(* CODESYS project Scheduler.project
   Company: Control Techniques
   Title: Scheduller
   Description: This program can be use to Start/stop motor  following  an weekly schedulle.  Up to 3 different time slices can be setup.
   Author: Angel Guerrero
   Version: 0.0.1

Project tree, tasks and I/O mapping:
  Drive : Unidrive M700, Nidec Control Techniques, version 1.8.0.9
    application Application
      Task Configuration
        Freewheeling
      program Freewheeling [ST]: TIMER, validate, get_vars, Initial
      function block Scheduler [ST]: Time_Check
      global variables GVL
      function Wait_Time [ST]
    RTEthernet
    Ethernet : Ethernet, Nidec Control Techniques, version 1.8.0.9
    <Empty>
    <Empty>
    <Empty>
  Advanced Link Editor
*)

// Drive/Application/GVL
{attribute 'qualified_only'}
VAR_GLOBAL
	RTC		 : DINT;  //RTC time from drive
	get_hr	 : UINT;  //Variable to hold hour 
	get_min	 : UINT;  //Variable to holf minutes [not used yet]
	get_sec	 : UINT;  //Variable that hold seconds [not used yet]
	get_wkd : SINT;  //Holds the week day
	enbl_mcr : INT;   //Enable Macro
END_VAR

// Drive/Application/Freewheeling
PROGRAM Freewheeling
VAR	
	err				: BOOL;			
	Scheduler_1		: Scheduler;
	Scheduler_2		: Scheduler;
	Scheduler_3		: Scheduler;	
	first_shoot		: BOOL := TRUE;	
END_VAR

//Version 0.00.01
//Angel Guerrero  Applications Engineer LatinAmerica July/2019
//============================================\\
get_vars();   	//Read RTC data
Initial();      //Macro setup
validate();   	//Validate setup data is correct
TIMER();        //Call the main program wich is timer.

ACTION TIMER:
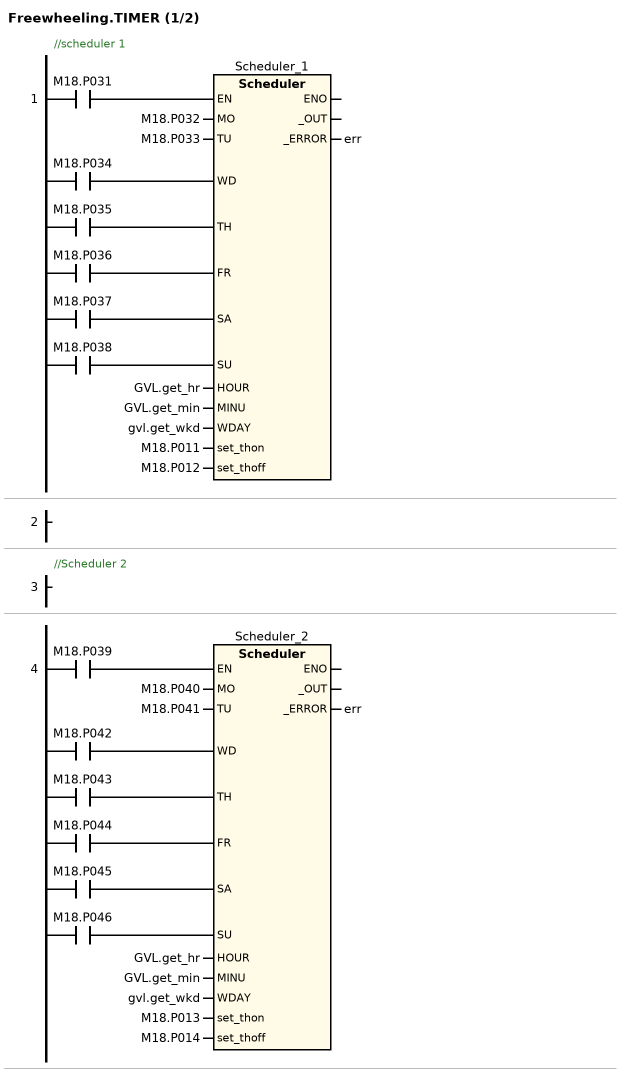
// NETWORK 1
// //scheduler 1
IF M18.P031 THEN
    Scheduler_1(
        MO := M18.P032,
        TU := M18.P033,
        WD := M18.P034,
        TH := M18.P035,
        FR := M18.P036,
        SA := M18.P037,
        SU := M18.P038,
        HOUR := GVL.get_hr,
        MINU := GVL.get_min,
        WDAY := gvl.get_wkd,
        set_thon := M18.P011,
        set_thoff := M18.P012,
        _ERROR => err); // Scheduler
END_IF

// NETWORK 2

// NETWORK 3
// //Scheduler 2

// NETWORK 4
IF M18.P039 THEN
    Scheduler_2(
        MO := M18.P040,
        TU := M18.P041,
        WD := M18.P042,
        TH := M18.P043,
        FR := M18.P044,
        SA := M18.P045,
        SU := M18.P046,
        HOUR := GVL.get_hr,
        MINU := GVL.get_min,
        WDAY := gvl.get_wkd,
        set_thon := M18.P013,
        set_thoff := M18.P014,
        _ERROR => err); // Scheduler
END_IF

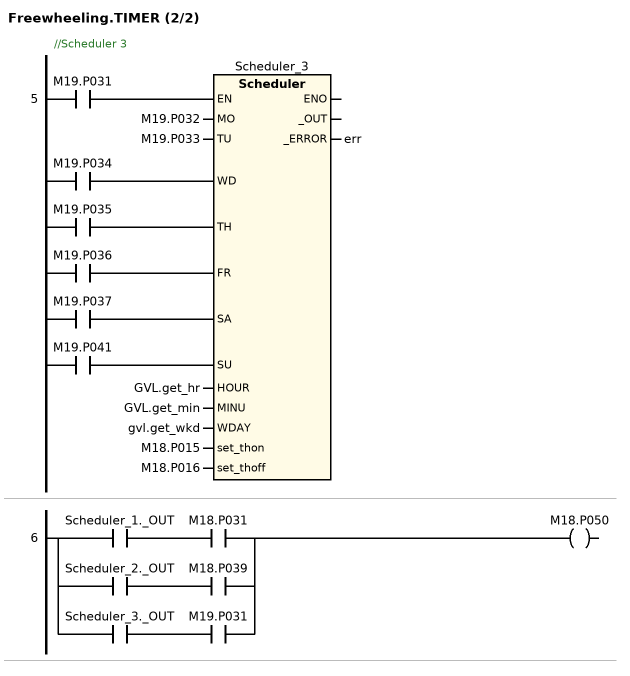
// NETWORK 5
// //Scheduler 3
IF M19.P031 THEN
    Scheduler_3(
        MO := M19.P032,
        TU := M19.P033,
        WD := M19.P034,
        TH := M19.P035,
        FR := M19.P036,
        SA := M19.P037,
        SU := M19.P041,
        HOUR := GVL.get_hr,
        MINU := GVL.get_min,
        WDAY := gvl.get_wkd,
        set_thon := M18.P015,
        set_thoff := M18.P016,
        _ERROR => err); // Scheduler
END_IF

// NETWORK 6
M18.P050 := Scheduler_1._OUT AND M18.P031 OR Scheduler_2._OUT AND M18.P039 OR Scheduler_3._OUT AND M19.P031;
END_ACTION

ACTION validate:
//Validate Scheduler 0 time ON/OFF is in correct range
IF M18.P011 >23 THEN
	M18.P011:=23;
END_IF
IF M18.P011 <0 THEN
	M18.P011:=0;
END_IF
//Validate Scheduler 0 time ON/OFF is in correct range
IF M18.P012 >23 THEN
	M18.P012:=23;
END_IF
IF M18.P012 <0 THEN
	M18.P012:=0;
END_IF
//Validate Scheduler 1 time ON/OFF is in correct range
IF M18.P013 >23 THEN
	M18.P013:=23;
END_IF
IF M18.P013 <0 THEN
	M18.P013:=0;
END_IF
//Validate Scheduler 1 time ON/OFF is in correct range
IF M18.P014 >23 THEN
	M18.P014:=23;
END_IF
IF M18.P014 <0 THEN
	M18.P014:=0;
END_IF
//Validate Scheduler 2 time ON/OFF is in correct range
IF M18.P015 >23 THEN
	M18.P015:=23;
END_IF
IF M18.P015 <0 THEN
	M18.P015:=0;
END_IF
//Validate Scheduler 2 time ON/OFF is in correct range
IF M18.P016 >23 THEN
	M18.P016:=23;
END_IF
IF M18.P016 <0 THEN
	M18.P016:=0;
END_IF
//Validate y Setup mode is 1 or 2 
IF M18.P030 >3 THEN
	M18.P030:=3;   //Remote Keypad
END_IF
IF M18.P030 <1 THEN
	M18.P030:=1;   //Local Keypad
END_IF
END_ACTION

ACTION get_vars:


gvl.RTC			:= M06.P017;                        			//Get time from RTC
gvl.get_hr  	:= DINT_TO_UINT(TRUNC(gvl.RTC/10000));  		//Get HRs
gvl.get_min 	:= DINT_TO_UINT((TRUNC(gvl.RTC/100)) MOD 100);  //Get Mins
gvl.get_sec 	:= DINT_TO_UINT((gvl.RTC) MOD 100);   			//seconds
gvl.enbl_mcr 	:= M18.P029;                                    // User Parameter to enter a "secret" value 1234  to deploy a Macro that prepare drive to link schduler output to Rfwd command
gvl.get_wkd     := M06.P018;                                    // get week day from Pr 06.P018
END_ACTION

ACTION Initial:
//macro to setup the  drive to start stop based on the scheduler
IF (gvl.enbl_mcr =1234 AND first_shoot=TRUE) THEN   	// If 1234 is set on Pr18.P029 then we accomodate drive parameters use the scheduller output for the rfwd command
	M08.P022	:=	0.00; 		//clear destination [default is M06.030] RunFwd
	M09.P004	:=	18.050;   	// Logic Fucntion 1 source1-->Asigns the Schduller ouput to the  funtion 
    M09.P006    :=  0.00;	    // Logic Function 1 Source 2-->we can probably get rid of this set to allow user add a DI to this source as way to stop the drive by any other condition
	M09.P007    :=  TRUE;       // Logic Function 1 Source 2 invert
	M09.P008    :=  FALSE;      // Logic Function 1 Output invert. 
	M09.P010    :=  6.030;      // Logic Funtion 1 Destination  set to Pr [6.030] RunFwd
	M10.P000	:=	1001;    	//Save Parameters
	M10.P038	:= 	100; 	 	//Reset Drive
	Wait_Time(T#400MS);         //Delay for 400ms after save and reset. 
	first_shoot := FALSE;       //Run this  section once once
	
END_IF

//Setup the source  to get the RTC from  Local Keypad or Remote .
//When mode is change user must save parameter manually and reset the drive
IF M18.P030=1 THEN 
	M06.P019:=4;     //M18.P030=4  Local Keypad
	ELSIF  M18.P030=2 THEN		
	M06.P019:=5;     // M18.P030= 5 get the time from the Remote Keypad
	ELSIF M18.P030=3 THEN
	M06.P019:=0;	 // M18.P030=3 allow  to set the realtime clock value
END_IF
END_ACTION

END_PROGRAM

// Drive/Application/Scheduler
FUNCTION_BLOCK Scheduler
VAR_INPUT
	MO			:BOOL	:=TRUE;  //[1] Enables hourly ON/OFF monday
	TU			:BOOL	:=TRUE;	 //[2] Enables hourly ON/OFF tuesday
	WD			:BOOL	:=TRUE;	 //[3] Enables hourly ON/OFF wednesday
	TH			:BOOL	:=TRUE;  //[4] Enables hourly ON/OFF thursday
	FR			:BOOL	:=TRUE;  //[5] Enables hourly ON/OFF friday
	SA			:BOOL	:=TRUE;  //[6] Enables hourly ON/OFF saturday
	SU			:BOOL	:=TRUE;  //[0] Enables hourly ON/OFF sunday 
	HOUR		:UINT;			 // Hour extracted from M06.P017 and set to -->gvl.get_hr
	MINU		:UINT;			 //Minutes extracted from M06.P017 ( Not used by now)
	WDAY		:SINT;           //Day of the week[0..6] (Should be linked to  M06.P018)
	set_thon	:UINT;           //Input to link  Pr in the application menu  to set hours to ON.
	set_thoff	:UINT;			 //Input to link  Pr in the application menu  to set hours to OFF.
END_VAR
VAR_OUTPUT
	_OUT		:BOOL;           //Output of the scheduler 
	_ERROR		:BOOL;           //error Output
END_VAR
VAR
	
END_VAR

//Version 0.00.01
//Angel Guerrero  July/2019

CASE WDAY OF             // WDAY is get from drive Pr6.018
	0   :               //sunday
	IF SU= TRUE THEN
		time_Check();
	END_IF	
	IF  NOT SU AND _OUT=TRUE THEN  
		_OUT:=FALSE; // Check if we are in current day and the output is true but the current day was selected in the scheduler
	END_IF	
	1   :               //Monday
    IF MO= TRUE THEN
		time_Check();
	END_IF
	IF  NOT MO AND _OUT=TRUE THEN
		_OUT:=FALSE; // Check if we are in current day and the output is true but the current day was selected in the scheduler
	END_IF
	2   :				//Tuesday
	IF TU= TRUE THEN
		time_Check();
	END_IF
	IF  NOT TU AND _OUT=TRUE THEN
		_OUT:=FALSE; // Check if we are in current day and the output is true but the current day was selected in the scheduler
	END_IF
	3	:				//Wednesday
	IF WD= TRUE THEN
		time_Check();
	END_IF
	IF  NOT WD AND _OUT=TRUE THEN
		_OUT:=FALSE; // Check if we are in current day and the output is true but the current day was selected in the scheduler
	END_IF	
	4	:				//Thursday
	IF TH= TRUE THEN
		time_Check();
	END_IF
	IF  NOT TH AND _OUT=TRUE THEN
		_OUT:=FALSE; // Check if we are in current day and the output is true but the current day was selected in the scheduler
	END_IF
	5	:				//Friday
	IF FR= TRUE THEN
		time_Check();
	END_IF
	IF  NOT FR AND _OUT=TRUE THEN
		_OUT:=FALSE; // Check if we are in current day and the output is true but the current day was selected in the scheduler
	END_IF
	
	6	:				//Saturday
	IF SA= TRUE THEN
		time_Check();
	END_IF
	IF  NOT SA AND _OUT=TRUE THEN
		_OUT:=FALSE; // Check if we are in current day and the output is true but the current day was selected in the scheduler
	END_IF
	ELSE
	_OUT:= FALSE;
END_CASE
 IF  NOT SU AND NOT MO AND NOT TU AND NOT WD AND NOT TH AND NOT FR AND NOT SA THEN
	 _OUT:= FALSE;
 END_IF

ACTION Time_Check:

//Version 0.00.01
//Angel Guerrero  July/2019

IF (HOUR>=0 AND HOUR <24) AND (MINU>=0 AND MINU<60) AND (set_thon>=0 AND set_thon<24) THEN
	
	IF set_thon=set_thoff THEN               // If hour on=hour off set ouput to false. 
		_OUT:=FALSE;
	END_IF	

  	IF  (set_thon < set_thoff) THEN       // If hr on < Hr off
		IF (HOUR>=set_thon AND  HOUR < set_thoff ) THEN
	 		_OUT:=TRUE;                   //set the ouput
	 		ELSIF (HOUR >=set_thoff AND HOUR <set_thon) THEN
	 		_OUT:=FALSE;                  //reset output
	 			
            ELSE 
          		_OUT:=FALSE;
			END_IF
	END_IF
  	
	
IF  (set_thon > set_thoff) THEN           // If time  to set On > time set off Ie Set on at 22h and set off at 10 am
		
	IF (HOUR>=set_thon AND HOUR <=23  ) THEN
	 		_OUT:=TRUE;
	 		
	ELSIF  (HOUR < set_thoff) THEN
			_OUT:=TRUE;			
	
	ELSIF (HOUR >=set_thoff AND HOUR <set_thon) THEN
	 		_OUT:=FALSE; 	 			 	   	
		
    ELSIF (HOUR < set_thon AND  HOUR >set_thoff) THEN
		_OUT:=FALSE;			
	END_IF 
	
END_IF
END_IF
END_ACTION

END_FUNCTION_BLOCK

// Drive/Application/Wait_Time
//Simple wait block used TO cause a delay in the middle OF a PROGRAM.
//Useful for allowing the drive parameters to update before trying to read other parameter.

//Version 0.00.01
//Cannon Melville
FUNCTION Wait_Time : BOOL
VAR_INPUT
	tDelayTime	: TIME;
END_VAR
VAR
	tEndTime	: TIME; 	
END_VAR

(*	 
	Editing the code in this function may result in limited support. 	 
*)

tEndTime	:= TIME() + tDelayTime;  // tiempo final = al tiempo actual + la demora que requiero 

WHILE TIME() < tEndTime DO            // entro en ciclo infinito mientras el tiempo actual  menor que el tiempo final ( demora x )
	Wait_Time	:= FALSE;             // variable wait time  es la salida de la funcion que esta en falso mientras estamos en espera.
END_WHILE

Wait_Time	:= TRUE;                 // variable de salida se hace verdadera cuando salimos del ciclo.

END_FUNCTION
